Fanuc KAREL source: compact_preamble.KL

PROGRAM KT00092
%NOLOCKGROUP
VAR
H1 : ARRAY[2] OF SHORT
R2:REAL
OUT:REAL
BEGIN
H1[1]=2
R2=3.0
OUT=((H1[1]) * R2)
END KT00092
